# EPICS substitutions: ek9000App/Db/EL4032.substitutions
file EL4032.template
{       pattern
        {
                TERMINAL,

        }
        {
        }
}
